// TIA Portal V20 export
DATA_BLOCK "SqlTdsReceive"   // DB8
TITLE = SqlTdsReceive
{ S7_Optimized_Access := 'TRUE'; DB_Accessible_From_OPC_UA := 'FALSE' }
AUTHOR : SIEMENS SUP Applications
VERSION : 3.0
// DB for holding the received data array of byte from a Tabular Data Stream (TDS) command to a SQL database
// stored: DBAccessibleFromOPCUA false, MemoryReserve 0
   VAR
      tdsTelegramArrayLength { ExternalAccessible := 'False'; ExternalVisible := 'False'; ExternalWritable := 'False'} : UDInt;   // number of Bytes received by TDS telegram and TRCV input
      tdsTelegramArray { ExternalAccessible := 'False'; ExternalVisible := 'False'; ExternalWritable := 'False'} : Array[0..9999] of Byte;   // array of Bytes of reconstructed TDS telegram
   END_VAR
BEGIN
END_DATA_BLOCK
